FUNCTION_BLOCK NotGate (* Negate the input Boolean value *)
  (* Standard: 61499-2 *)
  (* Version 1.0, 2008-11-09, Cheng Pang, The University of Auckland, Stable build. *)
  (* Compiler header: package fb.rt.pnp; *)
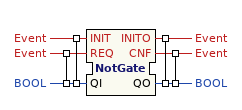
  EVENT_INPUT
    INIT WITH QI;
    REQ WITH QI; (* Normal Execution Request *)
  END_EVENT
  EVENT_OUTPUT
    INITO WITH QO;
    CNF WITH QO; (* Execution Confirmation *)
  END_EVENT
  VAR_INPUT
    QI : BOOL; (* Input event qualifier *)
  END_VAR
  VAR_OUTPUT
    QO : BOOL; (* Output event qualifier *)
  END_VAR
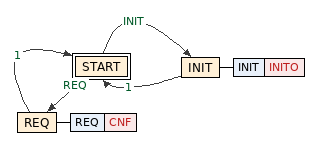
  EC_STATES
    START; (* Initial State *)
    REQ : REQ -> CNF; (* Normal execution *)
    INIT : INIT -> INITO;
  END_STATES
  EC_TRANSITIONS
    START TO REQ := REQ;
    REQ TO START := 1;
    START TO INIT := INIT;
    INIT TO START := 1;
  END_TRANSITIONS
  ALGORITHM REQ IN Java: (* Normally executed algorithm *)
if(QI.value){
  QO.value=false;
}
else{
  QO.value=true;
}
//System.out.println("  NotGate.REQ: ");
//System.out.println("QI.value = "+QI.value);
  END_ALGORITHM
  ALGORITHM INIT IN Java:
if(QI.value){
  QO.value=false;
}
else{
  QO.value=true;
}
//System.out.println("  NotGate.INIT: ");
//System.out.println("QI.value = "+QI.value);
  END_ALGORITHM
END_FUNCTION_BLOCK
